// TIA Portal V17 export
// export: Created 2025-06-26T07:49:57.5980111Z, ExportSetting WithDefaults, DisplayName Totally Integrated Automation Portal, DisplayVersion V17 Update 8, DisplayName TIA Portal Openness, DisplayVersion V17 Update 8, DisplayName TIA Portal Version Control Interface, DisplayVersion V17, DisplayName STEP 7 Professional, DisplayVersion V17 Update 8, DisplayName STEP 7 Safety, DisplayVersion V17 Update 6, DisplayName WinCC Advanced, DisplayVersion V17 Update 8
TYPE "CompressorData-STRUCT"
// stored: IsFailsafeCompliant false
   STRUCT
      CompressorTypeNumber : Int;
      Limits : Struct   // Kompressor Grenzwerte (Müssen noch definiert werden)
         p_CrankCase_Max : Real;   // kPa
         p_Oil_Min : Real;   // kPa
         n_Compressor_Max : Real;   // RPM
         T_Motor_Max : Real;   // C
         M_Motor_Limit : Real;   // %
         T_Inverter_Max : Real;   // C
      END_STRUCT;
      Constant : Struct   // Kompressor Konstanten (Müssen noch definiert werden)
         CompressionVolume_L : Real;
         CompressionLostPerPressureRatio : Real;
         PumpEfficinecy : Real;
      END_STRUCT;
      Settings : Bool;   // Kompressor Einstellungen (Müssen noch definiert werden)
   END_STRUCT;
END_TYPE
